Staubli VAL3: onExit.pgx

program onExit(bool x_bSaveInOut (dimensions=1), bool x_bsaveData (dimensions=1))
  local num l_nResult
  local string l_sMessage
begin
  // SAVE IT
  if x_bSaveInOut
    call out:save(l_nResult)
    if l_nResult!=0
      call language:message(l_sMessage,-6)
      popUpMsg(l_sMessage+toString("",l_nResult))
      logMsg("[KERNEL] INTERFACE:Error saving Out code: "+toString("",l_nResult))
    else
    endIf
    call in:save(l_nResult)
    if l_nResult!=0
      call language:message(l_sMessage,-6)
      popUpMsg(l_sMessage+toString("",l_nResult))
      logMsg("[KERNEL] INTERFACE:Error saving In code: "+toString("",l_nResult))
    endIf
    // save all the data
    if x_bsaveData
      l_nResult=saveData:libSave()
      if l_nResult!=0
        call language:message(l_sMessage,-6)
        popUpMsg(l_sMessage+toString("",l_nResult))
        logMsg("[KERNEL] INTERFACE:Error saving saveData code: "+toString("",l_nResult))
      endIf
    endIf
  endIf
  // clear the list
  call use:listempty()
end
